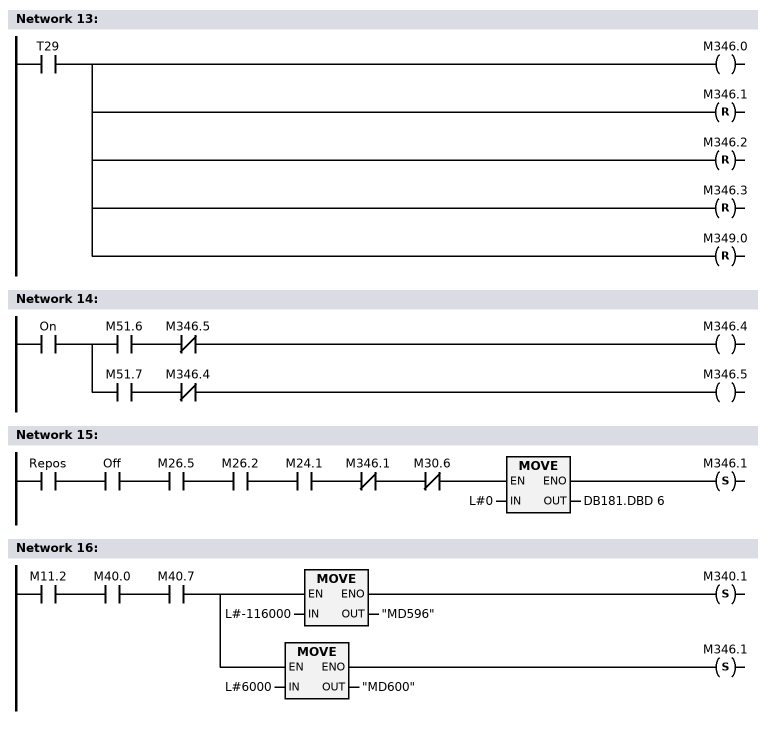
[picture p197: FC81 - GEST AXIS networks 13-16]
NETWORK
TITLE =
      A     "T29";
      =     "M346.0";
      R     "M346.1";
      R     "M346.2";
      R     "M346.3";
      R     "M349.0";
NETWORK
TITLE =
      A     "On";
      =     L 15.0;
      A     L 15.0;
      A     "M51.6";
      AN    "M346.5";
      =     "M346.4";
      A     L 15.0;
      A     "M51.7";
      AN    "M346.4";
      =     "M346.5";
NETWORK
TITLE =
      A     "Repos";
      A     "Off";
      A     "M26.5";
      A     "M26.2";
      A     "M24.1";
      AN    "M346.1";
      AN    "M30.6";
      JNB   M003;
      L     L#0;
      T     DB181.DBD 6;
      SET;
      SAVE;
      CLR;
M003: A     BR;
      S     "M346.1";
NETWORK
TITLE =
      A     "M11.2";
      A     "M40.0";
      A     "M40.7";
      =     L 15.0;
      A     L 15.0;
      JNB   M004;
      L     L#-116000;
      T     "MD596";
      SET;
      SAVE;
      CLR;
M004: A     BR;
      S     "M340.1";
      A     L 15.0;
      JNB   M005;
      L     L#6000;
      T     "MD600";
      SET;
      SAVE;
      CLR;
M005: A     BR;
      S     "M346.1";
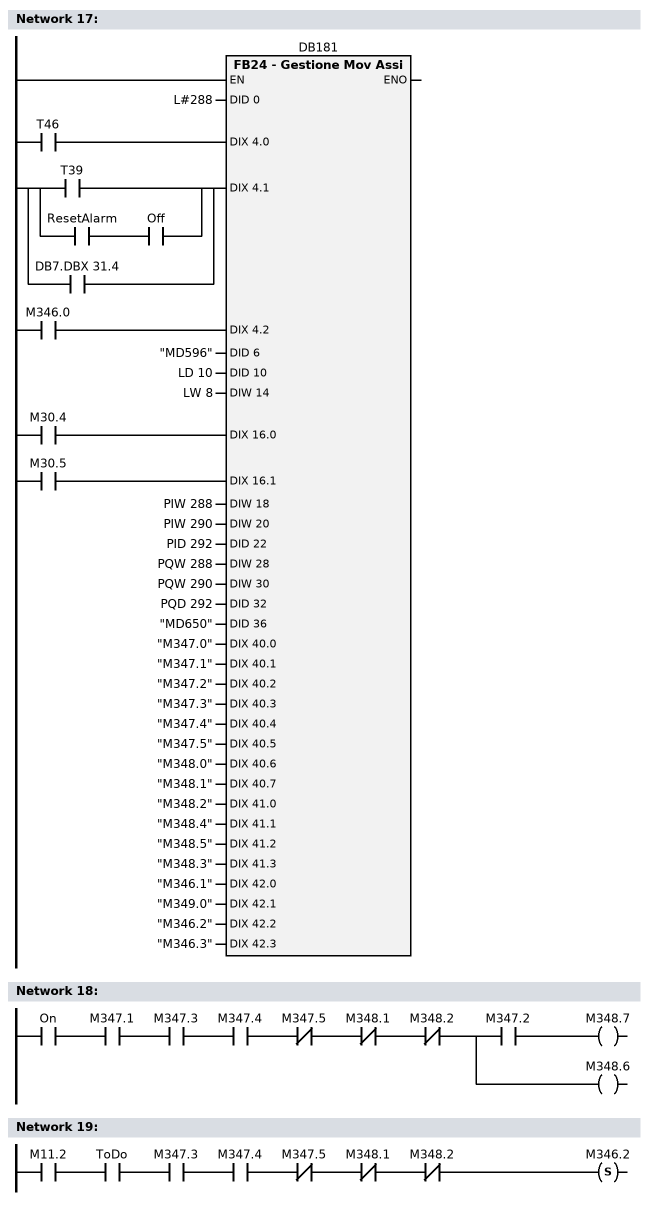
NETWORK
TITLE =
      A     "T46";
      =     L 15.0;
      BLD   103;
      A(;
      O     "T39";
      O;
      A     "ResetAlarm";
      A     "Off";
      O     DB7.DBX 31.4;
      );
      =     L 15.1;
      BLD   103;
      A     "M346.0";
      =     L 15.2;
      BLD   103;
      A     "M30.4";
      =     L 15.3;
      BLD   103;
      A     "M30.5";
      =     L 15.4;
      BLD   103;
      CALL  "FB24 - Gestione Mov Assi" , "DB181" (
           DID 0                    := L#288,
           DIX 4.0                  := L 15.0,
           DIX 4.1                  := L 15.1,
           DIX 4.2                  := L 15.2,
           DID 6                    := "MD596",
           DID 10                   := LD 10,
           DIW 14                   := LW 8,
           DIX 16.0                 := L 15.3,
           DIX 16.1                 := L 15.4,
           DIW 18                   := PIW 288,
           DIW 20                   := PIW 290,
           DID 22                   := PID 292,
           DIW 28                   := PQW 288,
           DIW 30                   := PQW 290,
           DID 32                   := PQD 292,
           DID 36                   := "MD650",
           DIX 40.0                 := "M347.0",
           DIX 40.1                 := "M347.1",
           DIX 40.2                 := "M347.2",
           DIX 40.3                 := "M347.3",
           DIX 40.4                 := "M347.4",
           DIX 40.5                 := "M347.5",
           DIX 40.6                 := "M348.0",
           DIX 40.7                 := "M348.1",
           DIX 41.0                 := "M348.2",
           DIX 41.1                 := "M348.4",
           DIX 41.2                 := "M348.5",
           DIX 41.3                 := "M348.3",
           DIX 42.0                 := "M346.1",
           DIX 42.1                 := "M349.0",
           DIX 42.2                 := "M346.2",
           DIX 42.3                 := "M346.3");
      NOP   0;
NETWORK
TITLE =
      A     "On";
      A     "M347.1";
      A     "M347.3";
      A     "M347.4";
      AN    "M347.5";
      AN    "M348.1";
      AN    "M348.2";
      =     L 15.0;
      A     L 15.0;
      A     "M347.2";
      =     "M348.7";
      A     L 15.0;
      BLD   102;
      =     "M348.6";
NETWORK
TITLE =
      A     "M11.2";
      A     "ToDo";
      A     "M347.3";
      A     "M347.4";
      AN    "M347.5";
      AN    "M348.1";
      AN    "M348.2";
      S     "M346.2";
END_FUNCTION

FUNCTION "FC117 - ERROR TOOL" : VOID	// FC 117
VERSION : 0.1
BEGIN
// (block stored without names or comments; labels and parameter names are numbered)
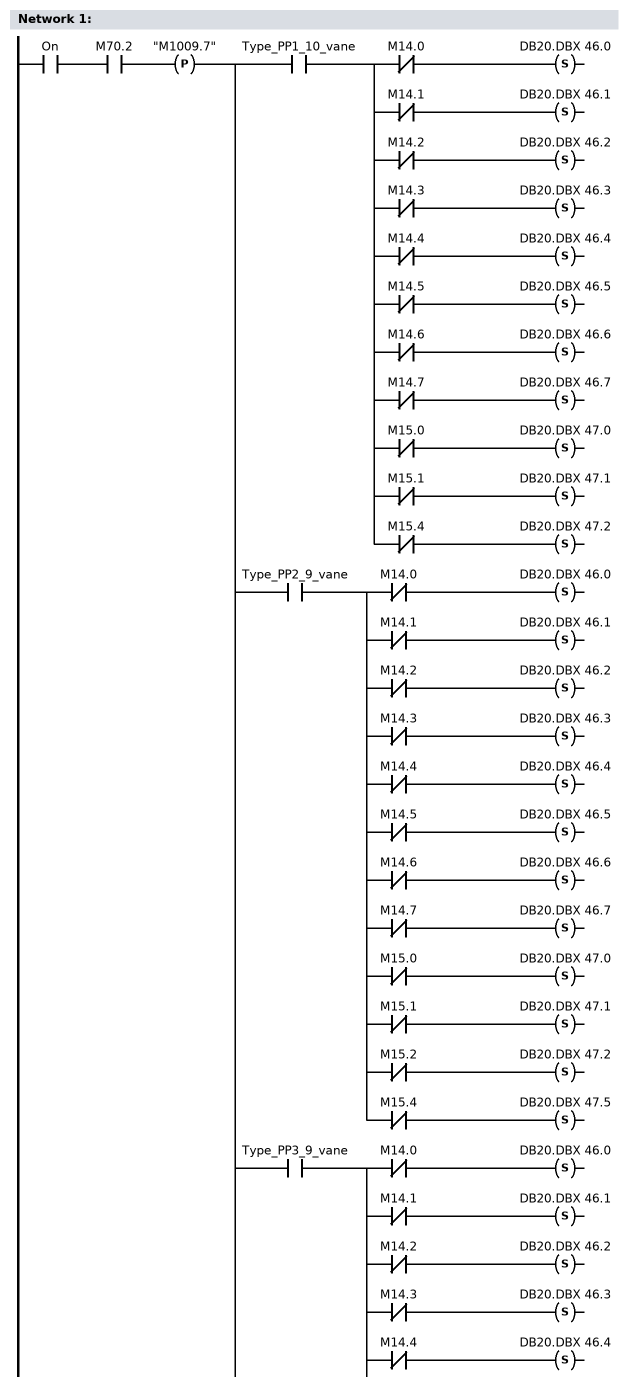
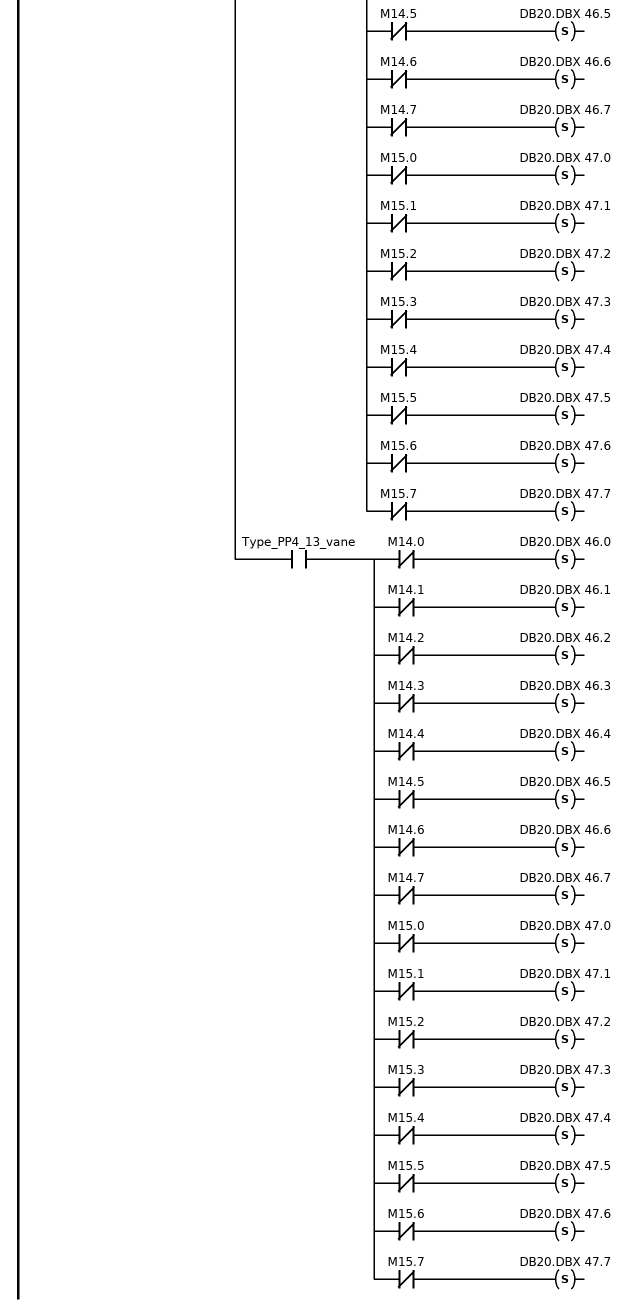
NETWORK
TITLE =
      A     "On";
      A     "M70.2";
      FP    "M1009.7";
      =     L 0.0;
      A     L 0.0;
      A     "Type_PP1_10_vane";
      =     L 0.1;
      A     L 0.1;
      AN    "M14.0";
      S     DB20.DBX 46.0;
      A     L 0.1;
      AN    "M14.1";
      S     DB20.DBX 46.1;
      A     L 0.1;
      AN    "M14.2";
      S     DB20.DBX 46.2;
      A     L 0.1;
      AN    "M14.3";
      S     DB20.DBX 46.3;
      A     L 0.1;
      AN    "M14.4";
      S     DB20.DBX 46.4;
      A     L 0.1;
      AN    "M14.5";
      S     DB20.DBX 46.5;
      A     L 0.1;
      AN    "M14.6";
      S     DB20.DBX 46.6;
      A     L 0.1;
      AN    "M14.7";
      S     DB20.DBX 46.7;
      A     L 0.1;
      AN    "M15.0";
      S     DB20.DBX 47.0;
      A     L 0.1;
      AN    "M15.1";
      S     DB20.DBX 47.1;
      A     L 0.1;
      AN    "M15.4";
      S     DB20.DBX 47.2;
      A     L 0.0;
      A     "Type_PP2_9_vane";
      =     L 0.1;
      A     L 0.1;
      AN    "M14.0";
      S     DB20.DBX 46.0;
      A     L 0.1;
      AN    "M14.1";
      S     DB20.DBX 46.1;
      A     L 0.1;
      AN    "M14.2";
      S     DB20.DBX 46.2;
      A     L 0.1;
      AN    "M14.3";
      S     DB20.DBX 46.3;
      A     L 0.1;
      AN    "M14.4";
      S     DB20.DBX 46.4;
      A     L 0.1;
      AN    "M14.5";
      S     DB20.DBX 46.5;
      A     L 0.1;
      AN    "M14.6";
      S     DB20.DBX 46.6;
      A     L 0.1;
      AN    "M14.7";
      S     DB20.DBX 46.7;
      A     L 0.1;
      AN    "M15.0";
      S     DB20.DBX 47.0;
      A     L 0.1;
      AN    "M15.1";
      S     DB20.DBX 47.1;
      A     L 0.1;
      AN    "M15.2";
      S     DB20.DBX 47.2;
      A     L 0.1;
      AN    "M15.4";
      S     DB20.DBX 47.5;
      A     L 0.0;
      A     "Type_PP3_9_vane";
      =     L 0.1;
      A     L 0.1;
      AN    "M14.0";
      S     DB20.DBX 46.0;
      A     L 0.1;
      AN    "M14.1";
      S     DB20.DBX 46.1;
      A     L 0.1;
      AN    "M14.2";
      S     DB20.DBX 46.2;
      A     L 0.1;
      AN    "M14.3";
      S     DB20.DBX 46.3;
      A     L 0.1;
      AN    "M14.4";
      S     DB20.DBX 46.4;
      A     L 0.1;
      AN    "M14.5";
      S     DB20.DBX 46.5;
      A     L 0.1;
      AN    "M14.6";
      S     DB20.DBX 46.6;
      A     L 0.1;
      AN    "M14.7";
      S     DB20.DBX 46.7;
      A     L 0.1;
      AN    "M15.0";
      S     DB20.DBX 47.0;
      A     L 0.1;
      AN    "M15.1";
      S     DB20.DBX 47.1;
      A     L 0.1;
      AN    "M15.2";
      S     DB20.DBX 47.2;
      A     L 0.1;
      AN    "M15.3";
      S     DB20.DBX 47.3;
      A     L 0.1;
      AN    "M15.4";
      S     DB20.DBX 47.4;
      A     L 0.1;
      AN    "M15.5";
      S     DB20.DBX 47.5;
      A     L 0.1;
      AN    "M15.6";
      S     DB20.DBX 47.6;
      A     L 0.1;
      AN    "M15.7";
      S     DB20.DBX 47.7;
      A     L 0.0;
      A     "Type_PP4_13_vane";
      =     L 0.1;
      A     L 0.1;
      AN    "M14.0";
      S     DB20.DBX 46.0;
      A     L 0.1;
      AN    "M14.1";
      S     DB20.DBX 46.1;
      A     L 0.1;
      AN    "M14.2";
      S     DB20.DBX 46.2;
      A     L 0.1;
      AN    "M14.3";
      S     DB20.DBX 46.3;
      A     L 0.1;
      AN    "M14.4";
      S     DB20.DBX 46.4;
      A     L 0.1;
      AN    "M14.5";
      S     DB20.DBX 46.5;
      A     L 0.1;
      AN    "M14.6";
      S     DB20.DBX 46.6;
      A     L 0.1;
      AN    "M14.7";
      S     DB20.DBX 46.7;
      A     L 0.1;
      AN    "M15.0";
      S     DB20.DBX 47.0;
      A     L 0.1;
      AN    "M15.1";
      S     DB20.DBX 47.1;
      A     L 0.1;
      AN    "M15.2";
      S     DB20.DBX 47.2;
      A     L 0.1;
      AN    "M15.3";
      S     DB20.DBX 47.3;
      A     L 0.1;
      AN    "M15.4";
      S     DB20.DBX 47.4;
      A     L 0.1;
      AN    "M15.5";
      S     DB20.DBX 47.5;
      A     L 0.1;
      AN    "M15.6";
      S     DB20.DBX 47.6;
      A     L 0.1;
      AN    "M15.7";
      S     DB20.DBX 47.7;
END_FUNCTION

FUNCTION "TimeOut" : VOID	// FC 800
AUTHOR : Cellini
FAMILY : GCLib
NAME : TimeOut
VERSION : 1.0
BEGIN
// (block stored without names or comments; labels and parameter names are numbered)
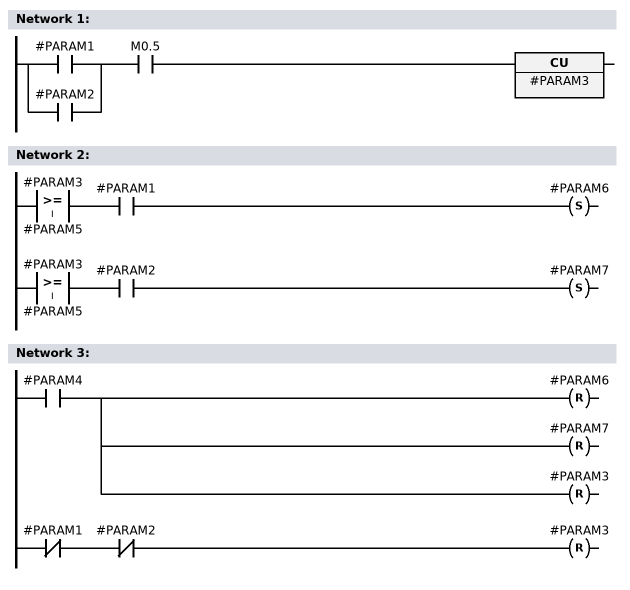
NETWORK
TITLE =
      A     #PARAM1;
      O     #PARAM2;
      A     "M0.5";
      CU    #PARAM3;
NETWORK
TITLE =
      L     #PARAM3;
      L     #PARAM5;
      >=I;
      A     #PARAM1;
      S     #PARAM6;
      L     #PARAM3;
      L     #PARAM5;
      >=I;
      A     #PARAM2;
      S     #PARAM7;
NETWORK
TITLE =
      A     #PARAM4;
      R     #PARAM6;
      R     #PARAM7;
      R     #PARAM3;
      AN    #PARAM1;
      AN    #PARAM2;
      R     #PARAM3;
END_FUNCTION

DATA_BLOCK "DI_Balluff1"	// DB 5
AUTHOR : Salvati
VERSION : 0.0
"BALLUFF"
BEGIN
END_DATA_BLOCK

DATA_BLOCK "DatiOP170B"	// DB 7
AUTHOR : Coletti
FAMILY : GCLib
VERSION : 0.1
BEGIN
// 382 bytes; values not shown
END_DATA_BLOCK

DATA_BLOCK DB 11
VERSION : 0.1
BEGIN
// 38 bytes; values not shown
END_DATA_BLOCK

DATA_BLOCK DB 12
VERSION : 0.1
BEGIN
// 38 bytes; values not shown
END_DATA_BLOCK

DATA_BLOCK DB 13
VERSION : 0.1
BEGIN
// 16 bytes; values not shown
END_DATA_BLOCK

DATA_BLOCK "Timer"	// DB 20
VERSION : 0.1
BEGIN
// 72 bytes; values not shown
END_DATA_BLOCK

DATA_BLOCK "DBWork"	// DB 21
AUTHOR : Coletti
VERSION : 0.1
BEGIN
// 478 bytes; values not shown
END_DATA_BLOCK

DATA_BLOCK "coordinate"	// DB 22
VERSION : 0.1
BEGIN
// 8860 bytes; values not shown
END_DATA_BLOCK

DATA_BLOCK DB 23
VERSION : 0.1
BEGIN
// 2 bytes; values not shown
END_DATA_BLOCK

DATA_BLOCK "DB180"	// DB 180
VERSION : 0.0
"FB24 - Gestione Mov Assi"
BEGIN
END_DATA_BLOCK

DATA_BLOCK "DB181"	// DB 181
VERSION : 0.0
"FB24 - Gestione Mov Assi"
BEGIN
END_DATA_BLOCK

ORGANIZATION_BLOCK "MAIN PROGRAM"	// OB 1
VERSION : 0.1
BEGIN
// (block stored without names or comments; labels and parameter names are numbered)
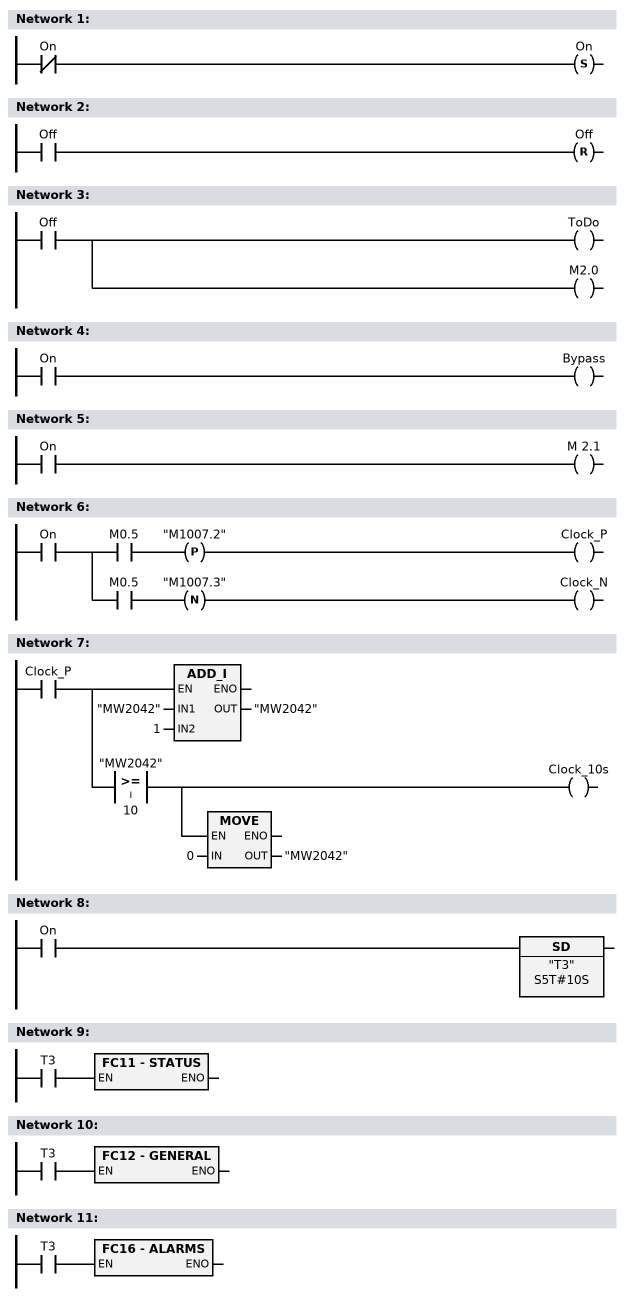
NETWORK
TITLE =
      AN    "On";
      S     "On";
NETWORK
TITLE =
      A     "Off";
      R     "Off";
NETWORK
TITLE =
      A     "Off";
      =     "ToDo";
      =     "M2.0";
NETWORK
TITLE =
      A     "On";
      =     "Bypass";
NETWORK
TITLE =
      A     "On";
      =     M 2.1;
NETWORK
TITLE =
      A     "On";
      =     L 20.0;
      A     L 20.0;
      A     "M0.5";
      FP    "M1007.2";
      =     "Clock_P";
      A     L 20.0;
      A     "M0.5";
      FN    "M1007.3";
      =     "Clock_N";
NETWORK
TITLE =
      A     "Clock_P";
      =     L 20.0;
      A     L 20.0;
      JNB   M001;
      L     "MW2042";
      L     1;
      +I;
      T     "MW2042";
M001: NOP   0;
      A     L 20.0;
      A(;
      L     "MW2042";
      L     10;
      >=I;
      );
      =     L 20.1;
      A     L 20.1;
      BLD   102;
      =     "Clock_10s";
      A     L 20.1;
      JNB   M002;
      L     0;
      T     "MW2042";
M002: NOP   0;
NETWORK
TITLE =
      A     "On";
      L     S5T#10S;
      SD    "T3";
NETWORK
TITLE =
      A     "T3";
      JNB   M003;
      CALL  "FC11 - STATUS";
M003: NOP   0;
NETWORK
TITLE =
      A     "T3";
      JNB   M004;
      CALL  "FC12 - GENERAL";
M004: NOP   0;
NETWORK
TITLE =
      A     "T3";
      JNB   M005;
      CALL  "FC16 - ALARMS";
M005: NOP   0;
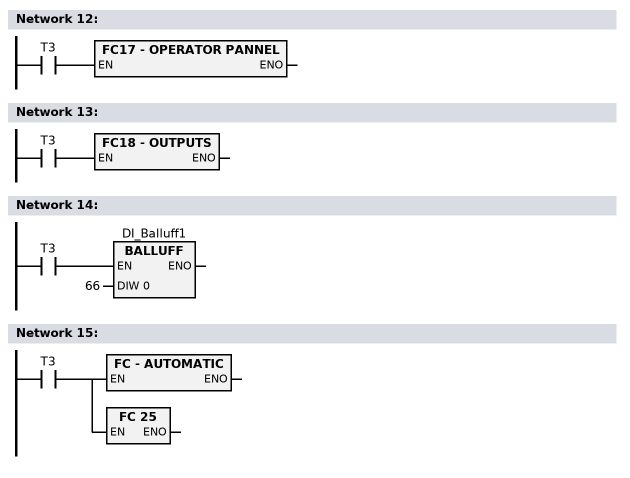
NETWORK
TITLE =
      A     "T3";
      JNB   M006;
      CALL  "FC17 - OPERATOR PANNEL";
M006: NOP   0;
NETWORK
TITLE =
      A     "T3";
      JNB   M007;
      CALL  "FC18 - OUTPUTS";
M007: NOP   0;
NETWORK
TITLE =
      A     "T3";
      JNB   M008;
      CALL  "BALLUFF" , "DI_Balluff1" (
           DIW 0                    := 66);
M008: NOP   0;
NETWORK
TITLE =
      A     "T3";
      =     L 20.0;
      A     L 20.0;
      JNB   M009;
      CALL  "FC - AUTOMATIC";
M009: NOP   0;
      A     L 20.0;
      JNB   M010;
      CALL  FC 25;
M010: NOP   0;
END_ORGANIZATION_BLOCK

ORGANIZATION_BLOCK "I/O_FLT1"	// OB 82
VERSION : 1.0
BEGIN
// (block stored without names or comments; labels and parameter names are numbered)
NETWORK
TITLE =
END_ORGANIZATION_BLOCK

ORGANIZATION_BLOCK "RACK_FLT"	// OB 86
VERSION : 0.1
BEGIN
// (block stored without names or comments; labels and parameter names are numbered)
NETWORK
TITLE =
END_ORGANIZATION_BLOCK

ORGANIZATION_BLOCK "COMPLETE RESTART"	// OB 100
VERSION : 0.1
BEGIN
// (block stored without names or comments; labels and parameter names are numbered)
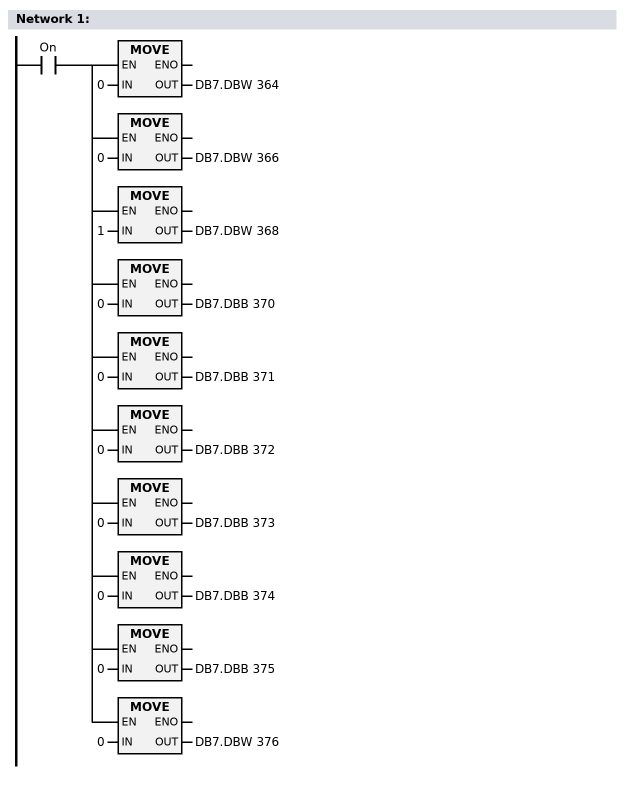
NETWORK
TITLE =
      A     "On";
      =     L 20.0;
      A     L 20.0;
      JNB   M001;
      L     0;
      T     DB7.DBW 364;
M001: NOP   0;
      A     L 20.0;
      JNB   M002;
      L     0;
      T     DB7.DBW 366;
M002: NOP   0;
      A     L 20.0;
      JNB   M003;
      L     1;
      T     DB7.DBW 368;
M003: NOP   0;
      A     L 20.0;
      JNB   M004;
      L     0;
      T     DB7.DBB 370;
M004: NOP   0;
      A     L 20.0;
      JNB   M005;
      L     0;
      T     DB7.DBB 371;
M005: NOP   0;
      A     L 20.0;
      JNB   M006;
      L     0;
      T     DB7.DBB 372;
M006: NOP   0;
      A     L 20.0;
      JNB   M007;
      L     0;
      T     DB7.DBB 373;
M007: NOP   0;
      A     L 20.0;
      JNB   M008;
      L     0;
      T     DB7.DBB 374;
M008: NOP   0;
      A     L 20.0;
      JNB   M009;
      L     0;
      T     DB7.DBB 375;
M009: NOP   0;
      A     L 20.0;
      JNB   M010;
      L     0;
      T     DB7.DBW 376;
M010: NOP   0;
END_ORGANIZATION_BLOCK

ORGANIZATION_BLOCK "MOD_ERR"	// OB 122
VERSION : 0.1
BEGIN
// (block stored without names or comments; labels and parameter names are numbered)
NETWORK
TITLE =
END_ORGANIZATION_BLOCK
